Staubli VAL3: check_plane.pgx

public program check_plane(tool x_tTool, bool& x_bCheck[])
  local point l_pPoint
begin
  //
  // CHECK IF THE TOOL IS INSIDE
  //
  x_bCheck=false
  //
  if bCreate_plane
    l_pPoint=here(x_tTool,fPlane)
    // check if inside
    if l_pPoint.trsf.z<=0.1
      // set to TRUE
      x_bCheck=true
    endIf
  endIf
end
